// TwinCAT 3 PLC project Untitled1
// ProgramVersion: 3.1.4026.1
// libraries:
//   Tc2_Standard, * (Beckhoff Automation GmbH)
//   Tc2_System, * (Beckhoff Automation GmbH)
//   Tc3_Module, * (Beckhoff Automation GmbH)
// project tree:
//   DUTs/ E_RtMode.TcDUT
//   / PlcTask.TcTTO
//   POUs/ FB_RtMode.TcPOU (not stored), FB_SetRtMode.TcPOU (not stored), FB_GetRtMode.TcPOU (not stored), F_UMRTAdvanceTick.TcPOU (not stored), F_UMRTGetTickMode.TcPOU, F_UMRTChangeTickMode.TcPOU (not stored), MAIN.TcPOU, MAIN_ExternalTick.TcPOU (not stored), MAIN_SelfTicks_F.TcPOU (not stored), MAIN_ExternalTick_ITc.TcPOU (not stored), MAIN_ExternalTick_F.TcPOU (not stored), MAIN_FastAsPossible.TcPOU (not stored), MAIN_FastAsPossible_ITc.TcPOU, MAIN_FastAsPossible_F.TcPOU (not stored)
// real-time tasks:
//   TASK PlcTask: cycle T#10ms, priority 20, ADS port 350

CONFIGURATION Untitled1
    RESOURCE PLC ON TwinCAT3
        TASK PlcTask(INTERVAL := T#10ms, PRIORITY := 20);
        PROGRAM MAIN WITH PlcTask : MAIN;
    END_RESOURCE
END_CONFIGURATION

// ---- DUTs/E_RtMode.TcDUT
{attribute 'qualified_only'}
{attribute 'strict'}
TYPE E_RtMode :  
(
	RtMode_Invalid := 16#FFFFFFFF,
	RtMode_FastAsPossible := 2,
	RtMode_Externaltick := 3,
	RtMode_Cyclic := 4
) UDINT;
END_TYPE

// ---- POUs/MAIN.TcPOU
PROGRAM MAIN
VAR
	fbrtmode : FB_RtMode; 
	n :DINT; 
END_VAR

n := n+1; 
//Using ADS
MAIN_ExternalTick(); 
MAIN_FastAsPossible();
 
//Using ITc
MAIN_ExternalTick_ITc(); 
MAIN_FastAsPossible_ITc(); 

//Using Functions 
MAIN_ExternalTick_F(); 
MAIN_SelfTicks_F(); 
MAIN_FastAsPossible_F();

END_PROGRAM

// ---- POUs/MAIN_FastAsPossible_ITc.TcPOU
PROGRAM MAIN_FastAsPossible_ITc
VAR
	
	fbRtmode : FB_RtMode; 
	state : INT := 0;	
	bStart : BOOL; 
	hr: HRESULT;
	eCurrentMode: E_RtMode;
END_VAR


VAR_OUTPUT 
	value AT %Q* : UDINT;	
END_VAR

hr := fbrtmode.ip.GetTickMode(eCurrentMode);

CASE state OF
	0:
		IF(bStart = TRUE) THEN 		
			state:= 1;
			value:=100; // steps to decrement as Cyclic 
		END_IF
	1:
		IF(eCurrentMode = E_RtMode.RtMode_Cyclic) THEN 
			value:=value-1; //decrementing Cyclic (near realtime speed) 
			IF value = 0 THEN
				state := 2;
				value:=100000; // Steps to decrement as a FastAsPossible 						
				(*switch to fastaspossible mode*)			
				fbRtmode.ip.ChangeTickMode(E_RtMode.RtMode_FastAsPossible);
			END_IF 	
		ELSE 
			state := 98; // ERROR 
		END_IF
	2:
		IF(eCurrentMode = E_RtMode.RtMode_FastAsPossible) THEN 
			value:=value-1; //decrementing as fast as possible 
			IF value = 0 THEN
				(*switch back to cyclic mode*)			
				state := 0;
				fbRtmode.ip.ChangeTickMode(E_RtMode.RtMode_Cyclic);			
			END_IF
		ELSE 
			state := 99; // ERROR 
		END_IF
END_CASE

END_PROGRAM

// ---- POUs/F_UMRTGetTickMode.TcPOU
FUNCTION F_UMRTGetTickMode : HRESULT
VAR_INPUT
	eMode : REFERENCE TO E_RtMode;
END_VAR

VAR
	ip : ITcRTimeSimulation;
END_VAR

F_UMRTGetTickMode := FW_ObjMgr_GetObjectInstance(oid:=16#02000000 (* Instance of RTIme*), iid:=TC_GLOBAL_IID_LIST.IID_ITcRTimeSimulation, pipUnk:=ADR(ip));
IF SUCCEEDED(F_UMRTGetTickMode) AND ip <> 0 THEN
	F_UMRTGetTickMode := ip.GetTickMode(eMode);
END_IF

END_FUNCTION
